Staubli VAL3: JointSpace.pjx

--- JointSpace.pjx ---
Parameters version=s7.9.1 stackSize=5000 millimeterUnit=true
Data file=JointSpace.dtx
Type name=JointPos path=./JointPos/JointPos.pjx
Type name=JointVel path=./JointVel/JointVel.pjx
Type name=JointAccel path=./JointAccel/JointAccel.pjx
Type name=JointForce path=./JointForce/JointForce.pjx

--- JointSpace.dtx ---
public JointPos jointPos
  [0]
    jointRx jp
public JointVel jointVel
  [0]
    num jv[6]
public JointAccel jointAccel
  [0]
    num ja[6]
public JointForce jointForce
  [0]
    num jf[6]
